// TIA Portal V17 export
// export: Created 2025-06-26T07:49:55.2553753Z, ExportSetting WithDefaults, DisplayName Totally Integrated Automation Portal, DisplayVersion V17 Update 8, DisplayName TIA Portal Openness, DisplayVersion V17 Update 8, DisplayName TIA Portal Version Control Interface, DisplayVersion V17, DisplayName STEP 7 Professional, DisplayVersion V17 Update 8, DisplayName STEP 7 Safety, DisplayVersion V17 Update 6, DisplayName WinCC Advanced, DisplayVersion V17 Update 8
TYPE "stHeartbeatCount2"
// stored: IsFailsafeCompliant false
   STRUCT
      nLocalCount : UInt;   // Count sent to remote partner
      nRemoteCount : UInt;   // Count received from remote partner
      bEnable : Bool;   // 1 = run heartbeat, 0 = disabled
      bOk : Bool;   // 1 = heatbeat ok, 0 = timeout
      nState : USInt;   // 0 = idle, 1 = ping, 2 = wait for pong, 3 = timeout
      tTimeout : Time := T#2s;   // Comm error timeout
   END_STRUCT;
END_TYPE
